TYPE sysInputs :
STRUCT
	
	
	iSwitch		 AT %I*: BOOL;

	iAlarmButton AT %I*: BOOL;
	
	iFacialDetec AT %I*: BOOL;
	iTestButton	 AT %I*: BOOL;
	
	iReedSwitch	 AT %I*: BOOL;
	iReedSwitch_rtrig : R_TRIG;
	
	
END_STRUCT
END_TYPE

(* stored: Version 1.1.0.1, ProductVersion 3.1.4026.18
   DUT sysInputs: Id {3a073515-8c62-4025-bb33-ff158228b7a2} *)
